// TIA Portal project "Foerderband" (V18)

(* hardware
DEVICE "S7-1500/ET200MP-Station_1"  S7-1500 station
   slot 0: "Profilschiene_0"  Rack  6ES7 590-1***0-0AA0
   slot 1: "Palettenlager01SPS"  CPU 1516-3 PN/DP  6ES7 516-3AN01-0AB0  V2.6
      slot 3: "CPU-Display_1"  6ES7591-1BA00-0AA0
      slot 32768: "PROFINET-Schnittstelle_1"  X1
         slot 32769: "Port_1"  X1 P1
         slot 32770: "Port_2"  X1 P2
      slot 33024: "PROFINET-Schnittstelle_2"  X2
         slot 33025: "Port_1"  X2 P1
      slot 33280: "DP-Schnittstelle_1"  X3
   slot 2: "AI 8xU/I/RTD/TC ST_1"  AI 8xU/I/RTD/TC ST  6ES7 531-7KF00-0AB0  V2.0
   slot 3: "AQ 4xU/I ST_1"  AQ 4xU/I ST  6ES7 532-5HD00-0AB0  V2.0
   slot 4: "DI 32x24VDC HF_1"  DI 32x24VDC HF  6ES7 521-1BL00-0AB0  V2.1
   slot 5: "DQ 32x24VDC/0.5A HF_1"  DQ 32x24VDC/0.5A HF  6ES7 522-1BL01-0AB0  V1.0
DEVICE "ET 200SP-Station_1"  ET 200SP-Station
   slot 0: "Baugruppenträger_0"  Rack  6ES5 710-8MAx1
   slot 0: "Palettenlager01DP"  IM 155-6 PN HF  6ES7 155-6AU00-0CN0  V3.3
   slot 1: "DI 8x24VDC HF_1"  DI 8x24VDC HF  6ES7 131-6BF00-0CA0  V2.0
      slot 1: "DI 8x24VDC HF_1"  DI 8x24VDC HF
   slot 2: "DQ 8x24VDC/0.5A HF_1"  DQ 8x24VDC/0.5A HF  6ES7 132-6BF00-0CA0  V2.0
      slot 1: "DQ 8x24VDC/0.5A HF_1"  DQ 8x24VDC/0.5A HF
   slot 3: "DI 8x24VDC HF_2"  DI 8x24VDC HF  6ES7 131-6BF00-0CA0  V2.0
      slot 1: "DI 8x24VDC HF_2"  DI 8x24VDC HF
   slot 4: "DQ 8x24VDC/0.5A HF_2"  DQ 8x24VDC/0.5A HF  6ES7 132-6BF00-0CA0  V2.0
      slot 1: "DQ 8x24VDC/0.5A HF_2"  DQ 8x24VDC/0.5A HF
   slot 5: "CM 4xIO-Link_1"  CM 4xIO-Link  6ES7 137-6BD00-0BA0  V2.1
      slot 1: "CM 4xIO-Link_1"  6ES7 137-6BD00-0BA0
   slot 6: "AI 2xU/I 2-/4-wire HS_1"  AI 2xU/I 2-,4-wire HS  6ES7 134-6HB00-0DA1  V1.1
      slot 1: "AI 2xU/I 2-/4-wire HS_1"  AI 2xU/I 2-,4-wire HS
   slot 7: "AI 2xU/I 2-/4-wire HS_2"  AI 2xU/I 2-,4-wire HS  6ES7 134-6HB00-0DA1  V1.1
      slot 1: "AI 2xU/I 2-/4-wire HS_2"  AI 2xU/I 2-,4-wire HS
   slot 8: "AQ 2xU/I HS_1"  AQ 2xU/I HS  6ES7 135-6HB00-0DA1  V1.1
      slot 1: "AQ 2xU/I HS_1"  AQ 2xU/I HS
   slot 9: "Servermodul_1"  Server module  6ES7 193-6PA00-0AA0  V1.1
      slot 1: "Servermodul_1"  Server module
   slot 127: "BA 2xRJ45"  BA 2xRJ45  6ES7 193-6AR00-0AA0  V0.0
      slot 1: "Port_1"  X1 P1 R  6ES7 193-6AR00-0AA0  V0.0
      slot 2: "Port_2"  X1 P2 R  6ES7 193-6AR00-0AA0  V0.0
DEVICE "HMI_1"  TP900 Comfort
   slot 0: "HMI_1"  TP900 Comfort  6AV2 124-0JC01-0AX0  16.0.0.0
   slot 1: "HMI_RT_1"  TP900 Comfort  6AV2 124-0JC01-0AX0  16.0.0.0
   slot 5: "HMI_1.IE_CP_1"  PROFINET Interface  16.0.0.0
      slot 1: "PROFINET Interface_1"  PROFINET Interface
         slot 1: "Port_1"  Port
         slot 2: "Port_2"  Port
   slot 7: "HMI_1.MPI/DP_CP_1"  MPI/DP Interface  16.0.0.0
*)

// ===== PLC "Palettenlager01SPS"  CPU 1516-3 PN/DP =====

VAR_GLOBAL   // PLC tag table "Standard-Variablentabelle"
   "System_Byte" AT %MB1 : Byte;
   "FirstScan" AT %M1.0 : Bool;
   "DiagStatusUpdate" AT %M1.1 : Bool;
   "AlwaysTRUE" AT %M1.2 : Bool;
   "AlwaysFALSE" AT %M1.3 : Bool;
   "Button_Board" AT %I30.0 : Bool;
   "BG2_Sensor" AT %I50.1 : Bool;   // Position of the right end of conveyor
   "BG6_Sensor" AT %I51.5 : Bool;   // Plunger bottom
   "BG7_Sensor" AT %I51.6 : Bool;   // Plunger middle
   "BG8_Sensor" AT %I51.7 : Bool;   // Plunger on top
   "Q_Motor_rotation" AT %Q50.6 : Bool;
   "Q_Plunger_Separator" AT %Q51.2 : Bool;
   "Q_Plunger_Down" AT %Q51.3 : Bool;
   "Q_Plunger_UP" AT %Q51.4 : Bool;
END_VAR

DATA_BLOCK "System_DB"   // DB1
{ S7_Optimized_Access := 'TRUE' }
VERSION : 0.1
// stored: InstanceOfName System
"System"
BEGIN
END_DATA_BLOCK

FUNCTION_BLOCK "Sequencer"   // FB1, FBD
{ S7_Optimized_Access := 'TRUE' }
VERSION : 0.1
   VAR_INPUT
      BG_2_Sensor : Bool;
      BG_6_Sensor : Bool;
      BG_7_Sensor : Bool;
      BG_8_Sensor : Bool;
      Start_Button : Bool;
      FirstScan : Bool;
   END_VAR
   VAR
      Step_0 : Bool;
      Step_1 : Bool;
      Step_2 : Bool;
      Step_3 : Bool;
      Step_4 : Bool;
      Step_5 : Bool;
      Step_6 : Bool;
      Step_7 : Bool;
   END_VAR
BEGIN

REGION Network 1: X_0
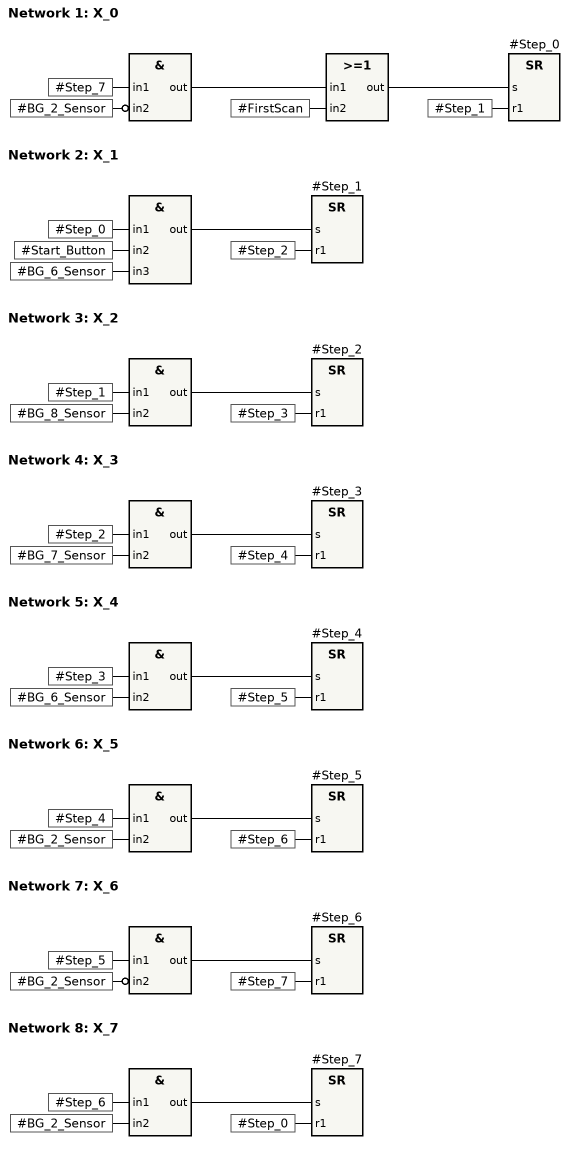
   IF (#Step_7 AND NOT #BG_2_Sensor) OR #FirstScan THEN
       #Step_0 := TRUE;   // SR flip-flop
   END_IF;
   IF #Step_1 THEN #Step_0 := FALSE; END_IF;
END_REGION

REGION Network 2: X_1
   IF #Step_0 AND #Start_Button AND #BG_6_Sensor THEN
       #Step_1 := TRUE;   // SR flip-flop
   END_IF;
   IF #Step_2 THEN #Step_1 := FALSE; END_IF;
END_REGION

REGION Network 3: X_2
   IF #Step_1 AND #BG_8_Sensor THEN
       #Step_2 := TRUE;   // SR flip-flop
   END_IF;
   IF #Step_3 THEN #Step_2 := FALSE; END_IF;
END_REGION

REGION Network 4: X_3
   IF #Step_2 AND #BG_7_Sensor THEN
       #Step_3 := TRUE;   // SR flip-flop
   END_IF;
   IF #Step_4 THEN #Step_3 := FALSE; END_IF;
END_REGION

REGION Network 5: X_4
   IF #Step_3 AND #BG_6_Sensor THEN
       #Step_4 := TRUE;   // SR flip-flop
   END_IF;
   IF #Step_5 THEN #Step_4 := FALSE; END_IF;
END_REGION

REGION Network 6: X_5
   IF #Step_4 AND #BG_2_Sensor THEN
       #Step_5 := TRUE;   // SR flip-flop
   END_IF;
   IF #Step_6 THEN #Step_5 := FALSE; END_IF;
END_REGION

REGION Network 7: X_6
   IF #Step_5 AND NOT #BG_2_Sensor THEN
       #Step_6 := TRUE;   // SR flip-flop
   END_IF;
   IF #Step_7 THEN #Step_6 := FALSE; END_IF;
END_REGION

REGION Network 8: X_7
   IF #Step_6 AND #BG_2_Sensor THEN
       #Step_7 := TRUE;   // SR flip-flop
   END_IF;
   IF #Step_0 THEN #Step_7 := FALSE; END_IF;
END_REGION
END_FUNCTION_BLOCK

FUNCTION_BLOCK "Sequencer_1"   // FB2, SCL
{ S7_Optimized_Access := 'TRUE' }
VERSION : 0.1
   VAR_INPUT
      BG_2_Sensor : Bool;
      BG_6_Sensor : Bool;
      BG_7_Sensor : Bool;
      BG_8_Sensor : Bool;
      Start_Button : Bool;
      FirstScan : Bool;
   END_VAR
   VAR
      Step_0 : Bool;
      Step_1 : Bool;
      Step_2 : Bool;
      Step_3 : Bool;
      Step_4 : Bool;
      Step_5 : Bool;
      Step_6 : Bool;
      Step_7 : Bool;
   END_VAR
BEGIN
   //Step 0
   IF (#Step_7 AND #BG_2_Sensor) OR #FirstScan THEN
       #Step_0:=TRUE;
   END_IF;

   IF #Step_1 THEN
       #Step_0 := FALSE;
   END_IF;

   //Step 1
   IF #Step_0 AND #BG_6_Sensor AND #Start_Button THEN
       #Step_1:= TRUE;
   END_IF;

   IF #Step_2 THEN
       #Step_1 := FALSE;
   END_IF;

   //Step 2
   IF #Step_1 AND #BG_8_Sensor THEN
       #Step_2 := TRUE;
   END_IF;

   IF #Step_3 THEN
       #Step_2 := FALSE;
   END_IF;

   //Step 3
   IF #Step_2 AND #BG_7_Sensor THEN
       #Step_3 := TRUE;
   END_IF;

   IF #Step_4 THEN
       #Step_3 := FALSE;
   END_IF;

   //Step 4
   IF #Step_3 AND #BG_6_Sensor THEN
       #Step_4 := TRUE;
   END_IF;

   IF #Step_5 THEN
       #Step_4 := FALSE;
   END_IF;

   //Step 5
   IF #Step_4 AND #BG_2_Sensor THEN
       #Step_5 := TRUE;
   END_IF;

   IF #Step_6 THEN
       #Step_5 := FALSE;
   END_IF;

   //Step 6
   IF #Step_5 AND #BG_2_Sensor THEN
       #Step_6 := TRUE;
   END_IF;

   IF #Step_7 THEN
       #Step_6 := FALSE;
   END_IF;

   //Step 7
   IF #Step_6 AND #BG_2_Sensor THEN
       #Step_7 := TRUE;
   END_IF;

   IF #Step_0 THEN
       #Step_7 := FALSE;
   END_IF;
END_FUNCTION_BLOCK

FUNCTION_BLOCK "System"   // FB3, FBD
{ S7_Optimized_Access := 'TRUE' }
VERSION : 0.1
   VAR_INPUT
      BG_2_Sensor : Bool;
      BG_6_Sensor : Bool;
      BG_7_Sensor : Bool;
      BG_8_Sensor : Bool;
      Start_Button : Bool;
      FirstScan : Bool;
   END_VAR
   VAR_OUTPUT
      Conveyor : Bool;
      Separator : Bool;
      Plunger_1_UP : Bool;
      Plunger_1_DOWN : Bool;
   END_VAR
   VAR
      Sequencer_Instance : "Sequencer";
      Outputs_Instance : "Outputs";
   END_VAR
BEGIN

REGION Network 1: Schrittkette
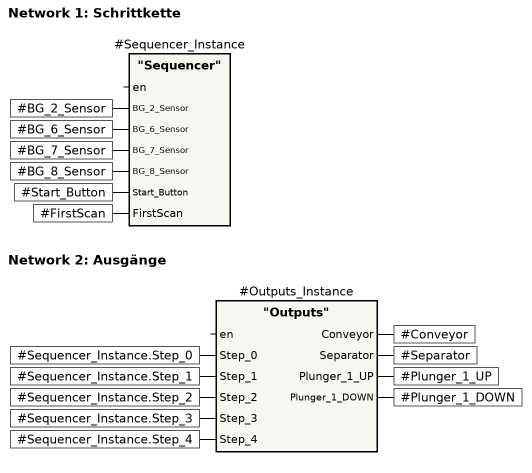
   #Sequencer_Instance(BG_2_Sensor := #BG_2_Sensor,   // "Sequencer"
                       BG_6_Sensor := #BG_6_Sensor,
                       BG_7_Sensor := #BG_7_Sensor,
                       BG_8_Sensor := #BG_8_Sensor,
                       Start_Button := #Start_Button,
                       FirstScan := #FirstScan);
END_REGION

REGION Network 2: Ausgänge
   #Outputs_Instance(Step_0 := #Sequencer_Instance.Step_0,   // "Outputs"
                     Step_1 := #Sequencer_Instance.Step_1,
                     Step_2 := #Sequencer_Instance.Step_2,
                     Step_3 := #Sequencer_Instance.Step_3,
                     Step_4 := #Sequencer_Instance.Step_4,
                     Conveyor => #Conveyor,
                     Separator => #Separator,
                     Plunger_1_UP => #Plunger_1_UP,
                     Plunger_1_DOWN => #Plunger_1_DOWN);
END_REGION
END_FUNCTION_BLOCK

FUNCTION_BLOCK "Outputs"   // FB4, SCL
{ S7_Optimized_Access := 'TRUE' }
VERSION : 0.1
   VAR_INPUT
      Step_0 : Bool;
      Step_1 : Bool;
      Step_2 : Bool;
      Step_3 : Bool;
      Step_4 : Bool;
   END_VAR
   VAR_OUTPUT
      Conveyor : Bool;
      Separator : Bool;
      Plunger_1_UP : Bool;
      Plunger_1_DOWN : Bool;
   END_VAR
BEGIN
   //#Conveyor ON/OFF
   IF #Step_4 THEN
       #Conveyor := true;
   END_IF;

   IF #Step_0 THEN
       #Conveyor := false;
   END_IF;

   //#Separator ON/OFF
   IF #Step_2 THEN
       #Separator := true;
   END_IF;

   IF #Step_0 OR #Step_3 THEN
       #Separator := false;
   END_IF;

   //#Plunger UP
   IF #Step_1 THEN
       #Plunger_1_UP := true;
   ELSE
       #Plunger_1_UP := False;
   END_IF;

   //#Plunger DOWN
   IF #Step_2 OR #Step_3 THEN
       #Plunger_1_DOWN := true;
   ELSE
       #Plunger_1_DOWN := False;
   END_IF;
END_FUNCTION_BLOCK

ORGANIZATION_BLOCK "Main"   // OB1, FBD, ProgramCycle
TITLE = "Main Program Sweep (Cycle)"
{ S7_Optimized_Access := 'TRUE' }
VERSION : 0.1
   VAR_INPUT
      Initial_Call : Bool;   // Initial call of this OB
      Remanence : Bool;   // =True, if remanent data are available
   END_VAR
BEGIN

REGION Network 1
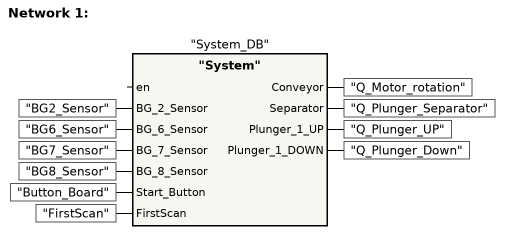
   "System_DB"(BG_2_Sensor := "BG2_Sensor",   // "System"
               BG_6_Sensor := "BG6_Sensor",
               BG_7_Sensor := "BG7_Sensor",
               BG_8_Sensor := "BG8_Sensor",
               Start_Button := "Button_Board",
               FirstScan := "FirstScan",
               Conveyor => "Q_Motor_rotation",
               Separator => "Q_Plunger_Separator",
               Plunger_1_UP => "Q_Plunger_UP",
               Plunger_1_DOWN => "Q_Plunger_Down");
END_REGION
END_ORGANIZATION_BLOCK

(* ===== HMI "HMI_RT_1" =====
system functions are stored by id; their names below are inferred from use
connection "HMI_Connection_1": ETHERNET, S7_1500_OMS

HMI tags "Default tag table"
   "Tag_ScreenNumber" : UInt, internal

text list "Textliste_Bildnamen": 1 'Root screen'

screen "Root screen" 800x420, template "Template_1"
   on GenerateScreen: SetTag("Tag_ScreenNumber", 1)
   Button "Button_1" at 29,25 size 96x32; TextOff 'Start'

Template "Template_1" 800x420
   Button "Beenden" at 720,360 size 78x58; TextOff 'Beenden'; PictureOff "ExitRuntime_TP900_Comfort_TR"; PictureOn "ExitRuntime_TP900_Comfort_TR"
      on Release: StopRuntime(0)
   Button "Template_Button" at 640,360 size 78x58; TextOff 'Text'
   Button "Template_Button_1" at 560,360 size 78x58; TextOff 'Text'
   Button "Template_Button_2" at 480,360 size 78x58; TextOff 'Text'
   Button "Template_Button_3" at 400,360 size 78x58; TextOff 'Text'
   Button "Template_Button_4" at 321,360 size 78x58; TextOff 'Text'
   Button "Template_Button_5" at 241,360 size 78x58; TextOff 'Text'
   Button "Template_Button_6" at 161,360 size 78x58; TextOff 'Text'
   Button "Meldungen" at 81,360 size 78x58; TextOff 'Meldungen'; PictureOff "AlarmDisplay_TP900_Comfort_TR"; PictureOn "AlarmDisplay_TP900_Comfort_TR"
      on Release: function_ef3f5d25("Alarm window_Unacknowledged", -1)
   Button "Startbild" at 1,360 size 78x58; TextOff 'Startbild'; PictureOff "NavigateHome_TP900_Comfort_TR"; PictureOn "NavigateHome_TP900_Comfort_TR"
      on Release: ActivateScreen("Root screen", 0)
*)